FUNCTION F_CounterNegativeOverflow : BOOL
VAR_INPUT
	COUNTERVALUE	: UINT;	
	ValueToSet		: REFERENCE TO UINT;
END_VAR
VAR
END_VAR

END_FUNCTION

(* stored: Version 1.1.0.1, ProductVersion 3.1.4024.11
   POU F_CounterNegativeOverflow: Id {92b9c22e-91a6-4220-928a-ec1733f656db}, SpecialFunc None *)
